// TIA Portal V19 export
VAR_GLOBAL   // PLC tag table "Default tag table"
   RETVAL_WWW AT %MW80 : Int;
   LampeStart AT %Q1.0 : Bool;
   Start_Stop AT %M10.0 : Bool;
   Compteur AT %MW2 : Int;
   PieceMax AT %MW100 : Int;
   "Compteur Bonnes Pièces" AT %MW10 : Int;
   "Compteur Mauvaises Pièces" AT %MW12 : Int;
   "Pointeur 1" AT %MD50 : DWord;
   "Pointeur 2" AT %MD54 : DWord;
   "A CHANGER" AT %MW200 : Word;
END_VAR
